PROGRAM P_Demo_FB_JsonDomParser_SetArray
VAR
    fbParser : FB_JsonDomParser; // 父 FB 实例
    v : SJsonValue;
    vRet : SJsonValue; // 返回值监视
    bTrigger : BOOL := FALSE; // 在线置 TRUE 触发一次调用
    bTriggerPrev : BOOL;
END_VAR

// =============================================================================
// 场景：修改已有 JSON 节点的 Array 类型值（如更新缓存的实时数据字段）。
// 价值：DOM 树本地修改不重新构造整个文档，比 GetDocument + 字符串替换效率高。
// 验证：登录 PLC 在线写 bTrigger := TRUE 触发，monitor 返回值/输出参数。具体步骤见下方注释。
// 验证步骤：
//   1. 右键 PLC 项目下 POUs 文件夹 → Add → Existing Item → 选本 .TcPOU 文件
//   2. 引用 Tc3_JsonXml（References → Add library）
//   3. 编译 → 登录 → 运行；按 verify 注释里给出的在线写值操作
// =============================================================================

// 上升沿触发一次方法调用并观察输出。
IF bTrigger AND NOT bTriggerPrev THEN
    vRet := fbParser.SetArray(
        v := v
    );
END_IF;
bTriggerPrev := bTrigger;

END_PROGRAM

(* stored: Version 1.1.0.1, ProductVersion 3.1.4024.5
   POU P_Demo_FB_JsonDomParser_SetArray: Id {6ec89e56-9792-5f57-b1a8-623c2fb39ea0}, SpecialFunc None *)
